// Mitsubishi GX Works2 project: WheelValveTurnFX0Test   PLC: FX0S/FX0

// global labels: Global1
VAR_GLOBAL
  Run AT M0 : BOOL;
  A2Toggle AT M20 : BOOL;
  ELToggle AT M30 : BOOL;
  ERToggle AT M40 : BOOL;
  A1N AT M11 : BOOL;
  A1P AT M12 : BOOL;
  A1Toggle AT M10 : BOOL;
  A2N AT M21 : BOOL;
  A2P AT M22 : BOOL;
  ELN AT M31 : BOOL;
  ELP AT M32 : BOOL;
  ERN AT M41 : BOOL;
  ERP AT M42 : BOOL;
  TurnFeedN AT M61 : BOOL;
  TurnFeedP AT M62 : BOOL;
  TurnFeed AT M60 : BOOL;
  RunI AT X000 : BOOL;
  RunStopI AT X001 : BOOL;
  RunIsManualI AT X002 : BOOL;
  A1PI AT X003 : BOOL;
  A2PI AT X004 : BOOL;
  ELNI AT X005 : BOOL;
  ELPI AT X006 : BOOL;
  ERNI AT X011 : BOOL;
  ERPI AT X012 : BOOL;
  A1ToggleO AT Y003 : BOOL;
  A2ToggleO AT Y004 : BOOL;
  ELToggleO AT Y005 : BOOL;
  ERToggleO AT Y006 : BOOL;
  TurnFeedO AT Y010 : BOOL;
  TurnFeedManual AT X015 : BOOL;
  TurnLock AT M50 : BOOL;
  TurnLockP AT M52 : BOOL;
  TurnLockO AT Y007 : BOOL;
  TurnLockN AT M51 : BOOL;
  RunIsManual AT M2 : BOOL;
  RunStop AT M1 : BOOL;
  RunStateFoil AT D1 : INT;
  RunState AT D0 : INT;
  TurnLockPI AT X007 : BOOL;
  TurnFeedPI AT X010 : BOOL;
END_VAR

// task Task_01 (event TRUE, interval 0, priority 31): POU_01

PROGRAM POU_01
VAR
  fRise : BOOL;
  fFall : BOOL;
  fTmp : BOOL;
  fELTouchFoil : BOOL;
  fRunStateNext : BOOL;
  fRunStateFoilNext : BOOL;
  fStepReady : BOOL;
  fTurnFeedDoneTimerEN : BOOL;
END_VAR
DECO(TRUE, RunState, 6, M100);
DECO(TRUE, RunStateFoil, 6, M200);
(*||||||||||||||||||||||||||||||||||||||||*)
(*  _____       _ _   _       _ _         *)
(* |_   _|     (_) | (_)     | (_)        *)
(*   | |  _ __  _| |_ _  __ _| |_ _______ *)
(*   | | | '_ \| | __| |/ _` | | |_  / _ \*)
(*  _| |_| | | | | |_| | (_| | | |/ /  __/*)
(* |_____|_| |_|_|\__|_|\__,_|_|_/___\___|*)
(*                                        *)
(*||||||||||||||||||||||||||||||||||||||||*)
RST(M8002, Run);
RST(M8002, RunStop);
RST(M8002, RunState); RST(M8002, RunStateFoil);
(*|||||||||||||||||||||||*)
(*  __  __       _       *)
(* |  \/  |     (_)      *)
(* | \  / | __ _ _ _ __  *)
(* | |\/| |/ _` | | '_ \ *)
(* | |  | | (_| | | | | |*)
(* |_|  |_|\__,_|_|_| |_|*)
(*                       *)
(*|||||||||||||||||||||||*)
SET(Run AND M100 AND M200, fTmp);
RST(fTmp, Run);
RST(fTmp, RunStop);
MOV(fTmp, 2, RunState); RST(fTmp, RunStateFoil);
RST(fTmp, fTmp);
SET(RunStop, fTmp);
RST(fTmp, RunStateFoil);
MOV(fTmp, 50, RunState);
RST(fTmp, fTmp);
(*|||||||||||||||||||||||||||||||||||||||||||||||||||||*)
(*  _                          _____ _             _   *)
(* | |                        / ____| |           | |  *)
(* | |     ___   ___  _ __   | (___ | |_ __ _ _ __| |_ *)
(* | |    / _ \ / _ \| '_ \   \___ \| __/ _` | '__| __|*)
(* | |___| (_) | (_) | |_) |  ____) | || (_| | |  | |_ *)
(* |______\___/ \___/| .__/  |_____/ \__\__,_|_|   \__|*)
(*                   | |                               *)
(*                   |_|                               *)
(*|||||||||||||||||||||||||||||||||||||||||||||||||||||*)
(*stop feed*)
SET(M102, fTmp);
RST(fTmp, TurnFeed);
SET(fTmp, fRunStateNext); RST(fTmp, fTmp);
(*stop feed done, eject foil*)
SET(M103 AND TurnFeedN, fTmp);
RST(fTmp, TurnLock);
SET(fTmp, fRunStateNext); RST(fTmp, fTmp);
(*eject foil done, start foil cycle*)
SET(M104 AND TurnLockN, fTmp);
MOV(fTmp, 2, RunStateFoil);
SET(fTmp, fRunStateNext); RST(fTmp, fTmp);
(*start foil cycle done, run loop*)
SET(M105 AND M205, fTmp);
MOV(fTmp, 10, RunStateFoil);
MOV(fTmp, 10, RunState);
RST(fTmp, fTmp);
(*|||||||||||||||||||||||||||||||||||||||||||||||||||||*)
(*|||||||||||||||||||||||||||||||||||||||||||||||||||||*)
(*move A1, A2, EL back*)
SET(M202, fTmp);
RST(fTmp, A1Toggle);
RST(fTmp, A2Toggle);
RST(fTmp, ELToggle);
SET(fTmp, fRunStateFoilNext); RST(fTmp, fTmp);
(*move A1, A2, EL back done, rotate ER back*)
SET(M203 AND A1N AND A2N AND ELN, fTmp);
RST(fTmp, ERToggle);
SET(fTmp, fRunStateFoilNext); RST(fTmp, fTmp);
(*rotate ER back done, wait*)
SET(M204 AND ERN, fTmp);
SET(fTmp, fRunStateFoilNext); RST(fTmp, fTmp);
(*||||||||||||||||||||||||||||||||||||||||||||||*)
(*  _                         _____             *)
(* | |                       |  __ \            *)
(* | |     ___   ___  _ __   | |__) |   _ _ __  *)
(* | |    / _ \ / _ \| '_ \  |  _  / | | | '_ \ *)
(* | |___| (_) | (_) | |_) | | | \ \ |_| | | | |*)
(* |______\___/ \___/| .__/  |_|  \_\__,_|_| |_|*)
(*                   | |                        *)
(*                   |_|                        *)
(*||||||||||||||||||||||||||||||||||||||||||||||*)
SET(Run AND RunIsManual, fStepReady);
SET(NOT RunIsManual, fStepReady);
(*rotate ER back done, move A1, A2 back*)
SET(fStepReady AND M210 AND ERN, fTmp);
RST(fTmp, A1Toggle);
RST(fTmp, A2Toggle);
SET(fTmp, fRunStateFoilNext); RST(fTmp, fTmp);
(*move A1, A2 back done, move EL forward half*)
SET(fStepReady AND M211 AND A1N AND A2N, fTmp);
SET(fTmp, ELToggle);
RST(fTmp, fELTouchFoil);
SET(fTmp, fRunStateFoilNext); RST(fTmp, fTmp);
(*move EL forward half done, move EL back*)
SET(fStepReady AND M212 AND fELTouchFoil, fTmp);
RST(fTmp, ELN);
RST(fTmp, ELToggle);
SET(fTmp, fRunStateFoilNext); RST(fTmp, fTmp);
(*move EL back done, rotate ER forward*)
SET(fStepReady AND M213 AND ELN, fTmp);
SET(fTmp, ERToggle);
SET(fTmp, fRunStateFoilNext); RST(fTmp, fTmp);
(*rotate ER forward done, wait*)
SET(fStepReady AND M214 AND ERP, fTmp);
MOV(fTmp, 20, RunStateFoil); RST(fTmp, fTmp);
(*move EL forward*)
SET(fStepReady AND M230, fTmp);
SET(fTmp, ELToggle);
SET(fTmp, fRunStateFoilNext); RST(fTmp, fTmp);
(*move EL forward done, move A1 forward*)
SET(fStepReady AND M231 AND ELP, fTmp);
SET(fTmp, A1Toggle);
SET(fTmp, fRunStateFoilNext); RST(fTmp, fTmp);
(*move A1 forward done, move EL back*)
SET(fStepReady AND M232 AND A1P, fTmp);
RST(fTmp, ELToggle);
SET(fTmp, fRunStateFoilNext); RST(fTmp, fTmp);
(*move EL back done, move A2 forward, rotate ER back*)
SET(fStepReady AND M233 AND ELN, fTmp);
SET(fTmp, A2Toggle);
RST(fTmp, ERToggle);
SET(fTmp, fRunStateFoilNext); RST(fTmp, fTmp);
(*move A2 forward done, wait*)
SET(fStepReady AND M234 AND A1P, fTmp);
MOV(fTmp, 40, RunStateFoil); RST(fTmp, fTmp);
(*||||||||||||||||||||||||||||||||||||||||||||||*)
(*||||||||||||||||||||||||||||||||||||||||||||||*)
(*run foil cycle at, wait command*)
SET(fStepReady AND M110 AND M220, fTmp);
MOV(fTmp AND RunIsManual AND Run, 30, RunStateFoil);
MOV(fTmp AND NOT RunIsManual, 30, RunStateFoil);
RST(fTmp, fTmp);
(*run foil cycle at, lock*)
SET(fStepReady AND M110 AND M240, fTmp);
SET(fTmp, TurnLock);
SET(fTmp, fRunStateNext); RST(fTmp, fTmp);
(*lock done, run foil cycle*)
OUT_T(TurnLockP, TC0, 2);
SET(fStepReady AND M111 AND TC0, fTmp);
MOV(fTmp, 10, RunStateFoil);
SET(fTmp, fRunStateNext); RST(fTmp, fTmp);
(*foil cycle at, feed*)
SET(fStepReady AND M112 AND M212, fTmp);
SET(fTmp, TurnFeed);
SET(fTmp, fRunStateNext); RST(fTmp, fTmp);
(*feed done, wait then end feed*)
OUT(TurnFeed AND TurnFeedPI, fTurnFeedDoneTimerEN);
OUT_T(fTurnFeedDoneTimerEN, TC1, 2);
SET(fStepReady AND M113 AND TC1, fTmp);
RST(fTmp, TurnFeedN);
RST(fTmp, TurnFeed);
RST(fTmp, fTurnFeedDoneTimerEN);
SET(fTmp, fRunStateNext); RST(fTmp, fTmp);
(*end feed done, eject foil*)
SET(fStepReady AND M114 AND TurnFeedN, fTmp);
RST(fTmp, TurnLock);
SET(fTmp, fRunStateNext); RST(fTmp, fTmp);
(*eject foil done, return*)
SET(fStepReady AND M115 AND TurnLockN, fTmp);
MOV(fTmp, 10, RunState); RST(fTmp, fTmp);
(**)
RST(fStepReady, fStepReady);

(**)
SET(M150, fTmp);
RST(fTmp, A1Toggle);
RST(fTmp, A2Toggle);
RST(fTmp, ELToggle);
RST(fTmp, TurnFeed);
INC(fTmp, RunState); RST(fTmp, fTmp);
SET(M151 AND A1N AND A2N AND ELN AND TurnFeedN, fTmp);
RST(fTmp, ERToggle);
RST(fTmp, TurnLock);
INC(fTmp, RunState); RST(fTmp, fTmp);
SET(M152 AND ERN AND TurnLockN, fTmp);
RST(fTmp, RunState);
RST(fTmp, RunStateFoil);
RST(fTmp, fTmp);
(**)
(*||||||||||||||*)
(*  _____ ____  *)
(* |_   _/ __ \ *)
(*   | || |  | |*)
(*   | || |  | |*)
(*  _| || |__| |*)
(* |_____\____/ *)
(*              *)
(*||||||||||||||*)
(*Input*)
OUT(NOT RunI, Run);
PLS(RunStopI, fRise); SET(fRise, RunStop);
OUT(RunIsManualI, RunIsManual);
PLS(A1PI, fRise); SET(fRise, A1P); RST(fRise, A1N);
PLS(A2PI, fRise); SET(fRise, A2P); RST(fRise, A2N);

(**)
(*PLS(ELNI, fRise); SET(fRise, ELN); RST(fRise, ELP);*)
(*PLS(ELPI, fRise); SET(fRise, ELP); RST(fRise, ELN);*)
PLS(ELPI, fRise); SET(fRise, ELN); RST(fRise, ELP); (*This is real ELN*)
PLS(ELNI, fRise); SET(fRise, ELP); RST(fRise, ELN); (*This is real ELP*)
(**)
PLS(ERNI, fRise); SET(fRise, ERN); RST(fRise, ERP);
PLS(ERPI, fRise); SET(fRise, ERP); RST(fRise, ERN);
PLS(TurnLockPI, fRise); SET(fRise, TurnLockP); RST(fRise, TurnLockN);
PLS(TurnFeedPI, fRise); SET(fRise, TurnFeedP); RST(fRise, TurnFeedN);
(*Output*)
OUT(A1Toggle, A1ToggleO);
OUT(A2Toggle, A2ToggleO);
OUT(ELToggle, ELToggleO);
OUT(ERToggle, ERToggleO);
OUT(TurnFeed, TurnFeedO);
OUT(TurnLock, TurnLockO);
SET(RunIsManual AND M100 AND TurnFeedManual, TurnFeed);
RST(RunIsManual AND M100 AND NOT TurnFeedManual, TurnFeed);
(*Input Cheat*)
OUT_T(NOT A1Toggle, TC2, 3); SET(TC2, A1N); RST(TC2, A1P);
OUT_T(NOT A2Toggle, TC3, 3); SET(TC3, A2N); RST(TC3, A2P);
OUT_T(NOT TurnLock, TC4, 5); SET(TC4, TurnLockN); RST(TC4, TurnLockP);
OUT_T(NOT TurnFeed, TC5, 5); SET(TC5, TurnFeedN); RST(TC5, TurnFeedP);
OUT_T(ELToggle, TC6, 5); SET(TC6, fELTouchFoil);
OUT_T(NOT ELToggle, TC7, 5); RST(TC7, fELTouchFoil);
(*Input Test)
OUT_T(Test AND A1Toggle, TC8, 10); SET(TC8, A1P); RST(TC8, A1N);
OUT_T(Test AND A2Toggle, TC9, 10); SET(TC9, A2P); RST(TC9, A2N);
OUT_T(Test AND ELToggle, TC10, 10); SET(TC10, ELP); RST(TC10, ELN);
OUT_T(Test AND NOT ELToggle, TC11, 10); SET(TC11, ELN); RST(TC11, ELP);
OUT_T(Test AND ERToggle, TC12, 10); SET(TC12, ERP); RST(TC12, ERN);
OUT_T(Test AND NOT ERToggle, TC13, 10); SET(TC13, ERN); RST(TC13, ERP);
OUT_T(Test AND TurnLock, TC14, 10); SET(TC14, TurnLockP); RST(TC14, TurnLockN);
OUT_T(Test AND TurnFeed, TC15, 10); SET(TC15, TurnFeedP); RST(TC15, TurnFeedN);
(**)
(*|||||||||||||||||||||||||||||||||||||||||||||||||||||||||||||||||||||||||||||||*)
(*|||||||||||||||||||||||||||||||||||||||||||||||||||||||||||||||||||||||||||||||*)
INC(fRunStateNext, RunState); RST(fRunStateNext, fRunStateNext);
INC(fRunStateFoilNext, RunStateFoil); RST(fRunStateFoilNext, fRunStateFoilNext);
END_PROGRAM
